FUNCTION_BLOCK SignalLightsController IMPLEMENTS ISignalLightsController
VAR
    _blinkTime : TIME := T#1000MS;
END_VAR

PROPERTY GetColorsSignalLightMachineModes :  ColorsSignalLightMachineModes
GET
END_GET
END_PROPERTY

PROPERTY GetColorsSignalLightMachineStatus : ColorsSignalLightMachineModes
GET
END_GET
END_PROPERTY

METHOD SetBlinkTime
VAR_INPUT
    blinkTime : TIME ;
END_VAR
_blinkTime := blinkTime;
END_METHOD

METHOD SetMachineMode : ColorsSignalLightMachineModes
VAR_INPUT
    currentMachineMode : eMachineModes := eMachineModes.Idle;
END_VAR
VAR_INST
    blinker : TP := (PT := _blinkTime);
END_VAR
IF eMachineModes.Home = currentMachineMode THEN
    blinker(in := TRUE);
ELSE
    blinker(in := FALSE);
END_IF

CASE currentMachineMode OF
    eMachineModes.Fault:
        SetMachineMode.Red    := TRUE;
        SetMachineMode.Green  := FALSE;
        SetMachineMode.Yellow := FALSE;

    eMachineModes.Idle:

        SetMachineMode.Red    := FALSE;
        SetMachineMode.Green  := FALSE;
        SetMachineMode.Yellow := FALSE;

    eMachineModes.Automat:
        SetMachineMode.Red    := FALSE;
        SetMachineMode.Green  := TRUE;
        SetMachineMode.Yellow := FALSE;

    eMachineModes.Step:
        SetMachineMode.Red    := FALSE;
        SetMachineMode.Green  := TRUE;
        SetMachineMode.Yellow := TRUE;

    eMachineModes.Home:
        SetMachineMode.Red    := FALSE;
        SetMachineMode.Yellow := FALSE;

        IF blinker.Q THEN
            SetMachineMode.Green := TRUE;
        ELSE
            SetMachineMode.Green := FALSE;
        END_IF

    eMachineModes.Manual:
        SetMachineMode.Red    := FALSE;
        SetMachineMode.Yellow := TRUE;
        SetMachineMode.Green  := FALSE;
ELSE
    ;
END_CASE
END_METHOD

METHOD SetMachineStatusOff : ColorsSignalLightsStatus
VAR_INPUT
    currentMachineStatus : eMachineStatus ;
END_VAR
END_METHOD

METHOD SetMachineStatusOn : ColorsSignalLightsStatus
VAR_INPUT
    currentMachineStatus	: eMachineStatus ;
END_VAR
END_METHOD

END_FUNCTION_BLOCK

(* stored: Version 1.1.0.1, ProductVersion 3.1.4024.12
   POU SignalLightsController: Id {a3831b7a-f468-072b-07bc-5d866e7a1270}, SpecialFunc None
   Property GetColorsSignalLightMachineModes: Id {ea4c7eb4-63fe-0480-14d4-dbd32e8f6cf8}
   Get Get: Id {4c4c40b2-ca35-01b0-3798-833f40d42b14}
   Property GetColorsSignalLightMachineStatus: Id {61c67baa-eee7-034d-2319-e69b1ea0ec47}
   Get Get: Id {337c6540-7a18-09a7-100a-9a6284d2aaa7}
   Method SetBlinkTime: Id {0da11680-2f5f-0252-3b6c-0817468bf029}
   Method SetMachineMode: Id {3a4f1b80-1872-04a2-0d9a-630ebf80f85e}
   Method SetMachineStatusOff: Id {b8bada96-3e7b-0287-112f-dcc29f5c588f}
   Method SetMachineStatusOn: Id {ac3547ba-4fce-0714-2ddd-7a82bdb7e26d} *)
